Fanuc KAREL source: kx00020.KL

PROGRAM KX00020
%STACKSIZE=65535
%PRIORITY=65535
%NOLOCKGROUP
VAR
I : INTEGER
J : INTEGER
B : BOOLEAN
F : FILE
S : STRING[80]
P : XYZWPR
SA : ARRAY[4] OF STRING[12]
BEGIN
-- UNRESOLVED_PC line 12 opcodes [3F 22 9D 33 61] marker_code=0
-- UNRESOLVED_PC line 13 opcodes [22 9D 33 5E 75] marker_code=17
END KX00020
